// TIA Portal V16 export
// export: Created 2021-09-08T12:46:13.4170587Z, ExportSetting WithDefaults, DisplayName Totally Integrated Automation Portal, DisplayVersion V16 Update 3, DisplayName TIA Portal Version Control Interface, DisplayVersion V16 Update 2, DisplayName TIA Portal Openness, DisplayVersion V16 Update 3, DisplayName TIA Portal Teamcenter Gateway, DisplayVersion V16, DisplayName STEP 7 Professional, DisplayVersion V16 Update 3, DisplayName STEP 7 Safety, DisplayVersion V16, DisplayName WinCC Advanced, DisplayVersion V16 Update 3
DATA_BLOCK "dbVolumeCounters"   // DB109
{ S7_Optimized_Access := 'FALSE' }
VERSION : 0.1
// stored: AutoNumber true, DBAccessibleFromOPCUA true, IsOnlyStoredInLoadMemory false, IsWriteProtectedInAS false
   VAR RETAIN
      FM201 : "FREQ_COUNTER";   // Витрата вхідної води FM201
      FM501 : "FREQ_COUNTER";   // Витрата вхідної води UF FM501
      FM502 : "FREQ_COUNTER";   // Витрата вхідної води UF FM502
      FM901 : "FREQ_COUNTER";   // Витрата пермеату RO FM901
      FM902 : "FREQ_COUNTER";   // Витрата концентрату RO FM902
      FM1201 : "FREQ_COUNTER";   // Витрата пермеату на споживоча FM1201
      FM1301 : "FREQ_COUNTER";   // Витрата пермеату NF FM1301
      FM1302 : "FREQ_COUNTER";   // Витрата концентрату NF FM1302
      FM1701 : "FREQ_COUNTER";   // Витрата нанофільтрату на споживоча FM1701
      FM1801 : "FREQ_COUNTER";   // Витрата стічних вод FM1801
   END_VAR
BEGIN
END_DATA_BLOCK
